{attribute addProperty BoxType "KL3351"}
{attribute addProperty Id "StatusAT %I*USINT000Ud_RegInAT %I*INT000UrefAT %I*INT000CtrlAT %Q*USINT000RegOutAT %Q*INT000"}
{attribute addProperty CRC "659443344"}
{attribute addProperty SizeInBites "0"}
{attribute addProperty SizeInBytes "0"}
TYPE Channel_274E4E90 :
STRUCT
	{attribute addProperty Name "Status"}
	Status AT %I* : USINT;
	{attribute addProperty Name "Ud_RegIn"}
	Ud_RegIn AT %I* : INT;
	{attribute addProperty Name "Uref"}
	Uref AT %I* : INT;
	{attribute addProperty Name "Ctrl"}
	Ctrl AT %Q* : USINT;
	{attribute addProperty Name "RegOut"}
	RegOut AT %Q* : INT;
END_STRUCT
END_TYPE

(* stored: Version 1.2.0.0, ProductVersion 3.1.4024.9
   DUT Channel_274E4E90: Id {bc99ac71-1d33-43af-a717-e817abf76404} *)
